{attribute 'GeneratedUsingTerminal: EPP6090-0000-0017'}
{attribute addProperty BoxType "EPP6090-0000-0017"}
{attribute addProperty Id "UpBOOL1DownBOOL1LeftBOOL1RightBOOL1EnterBOOL1TxPDO_ToggleBOOL1"}
{attribute addProperty CRC "3823631634"}
{attribute addProperty Size "6"}
TYPE Status_E3E7FD12 :
STRUCT
	{attribute addProperty Name "Up"}
	Up : BOOL;
	{attribute addProperty Name "Down"}
	Down : BOOL;
	{attribute addProperty Name "Left"}
	Left : BOOL;
	{attribute addProperty Name "Right"}
	Right : BOOL;
	{attribute addProperty Name "Enter"}
	Enter : BOOL;
	{attribute addProperty Name "TxPDO_Toggle"}
	TxPDO_Toggle : BOOL;
END_STRUCT
END_TYPE

(* stored: Version 1.2.0.0, ProductVersion 3.1.4024.9
   DUT Status_E3E7FD12: Id {f84f3f17-f3ba-482a-94a4-6bcfecb9ea62} *)
